PROGRAM PRG2_Object_Detectie
VAR
    ObjectAanwezig : BOOL;    			// Invoer van de sensor, TRUE als object gedetecteerd
    AlarmStatus    : BOOL;    			// Uitvoer, TRUE als er geen object is gedetecteerd
    MaxWachttijd   : TIME := T#5M;    	// Maximale tijd om te wachten op een object
    Wachttijd      : TIME;    			// Huidig wachttijd zonder objectdetectie
END_VAR



// lezen ingangen
ObjectAanwezig := GVL.LS_001; 

//reset wachttijd met alarm acknowledge
IF GVL.KN_002 THEN
	Wachttijd := T#0S;
	AlarmStatus := FALSE;
	GVL.PRG1_Status := 1;
END_IF


IF GVL.PRG1_Status = 1 THEN
	// Controleer of een object aanwezig is op de transportband
	IF ObjectAanwezig = TRUE THEN
		// Object gedetecteerd, reset de wachttijd en schakel het alarm uit
		Wachttijd := T#0S;
		AlarmStatus := FALSE;
	ELSE//wacht op detectie, tot maximale tijd verstreken en alarm geactiveerd
		// Geen object gedetecteerd, verhoog de wachttijd
			
		Wachttijd := Wachttijd + GVL.cyclusTijd;  // Verhoog de gewachtte tijd per cyclus 
	
		// Activeer het alarm als de wachttijd de maximale tijd overschrijdt
		IF Wachttijd >= MaxWachttijd THEN
			AlarmStatus := TRUE;
		END_IF
	END_IF
END_IF


//stuur statussen naar GVL.
GVL.objectDetected  :=  ObjectAanwezig;	
GVL.ALM001 			:= 	AlarmStatus; 	// schrijven in geheugen voor OPC/SCADA of weet ik het wat nog meer.
GVL.alarmActief 	:= 	AlarmStatus;	// sturen naar digitale uitgang

END_PROGRAM

(* stored: Version 1.1.0.1, ProductVersion 3.1.4024.12
   POU PRG2_Object_Detectie: Id {582db3f0-3a0b-4d59-91c1-6e5fa4d01714}, SpecialFunc None *)
